TYPE ST_ParamFixed :
STRUCT
END_STRUCT
END_TYPE

(* stored: Version 1.1.0.1, ProductVersion 3.1.4020.6
   DUT ST_ParamFixed: Id {727b2490-7f07-4554-8c32-6bd72c5b4e76} *)
